TYPE EM_CanSupply_ALM :
STRUCT
END_STRUCT
END_TYPE

(* stored: Version 1.1.0.1, ProductVersion 3.1.4024.12
   DUT EM_CanSupply_ALM: Id {b57ec392-0272-42f3-85e4-e9c43acaeca7} *)
